// TIA Portal V18 export
// export: Created 2026-06-23T03:11:38.3968089Z, ExportSetting WithDefaults, DisplayName Totally Integrated Automation Portal, DisplayVersion V18, DisplayName TIA Portal Openness, DisplayVersion V18, DisplayName TIA Portal Version Control Interface, DisplayVersion V18, DisplayName STEP 7 Professional, DisplayVersion V18, DisplayName STEP 7 Safety, DisplayVersion V18, DisplayName WinCC Professional, DisplayVersion V18
Screen "Screen_1"  1440x900, Number=2
  ScreenLayer 
    GraphicView "Graphic view_1" at 0,0 size 1440x900  Picture=Thiết kế chưa có tên (2)_1
    GraphicIOField "Graphic I/O field_9" at 430,521 size 275x288  Mode=Output, OnValue=1, PictureList=GL_BonChua_MucDich
      ProcessValue := HMI_Anim_BonChua1_MucDich
    GraphicIOField "Graphic I/O field_10" at 154,90 size 233x295  Mode=Output, OnValue=1, PictureList=GL_BonTron_MucDich
      ProcessValue := HMI_Anim_Bon1_MucDich
    GraphicIOField "Graphic I/O field_2" at 904,517 size 275x288  Mode=Output, OnValue=1, PictureList=GL_BonChua_MucDich
      ProcessValue := HMI_Anim_BonChua2_MucDich
    GraphicIOField "Graphic I/O field_3" at 486,90 size 233x295  Mode=Output, OnValue=1, PictureList=GL_BonTron_MucDich
      ProcessValue := HMI_Anim_Bon2_MucDich
    GraphicIOField "Graphic I/O field_4" at 811,89 size 233x295  Mode=Output, OnValue=1, PictureList=GL_BonTron_MucDich
      ProcessValue := HMI_Anim_Bon4_MucDich
    GraphicIOField "Graphic I/O field_6" at 1160,89 size 233x295  Mode=Output, OnValue=1, PictureList=GL_BonTron_MucDich
      ProcessValue := HMI_Anim_Bon3_MucDich
    GraphicView "Graphic view_3" at 201,61 size 11x113  Picture=Graphic_24
    GraphicIOField "Graphic I/O field_5" at 189,70 size 51x78  Mode=Output, OnValue=1, PictureList=GL_Van_NamDoc
      ProcessValue := V3230_Nuoc_Bon1
    GraphicView "Graphic view_2" at 544,60 size 11x113  Picture=Graphic_24
    GraphicIOField "Graphic I/O field_12" at 533,70 size 51x78  Mode=Output, OnValue=1, PictureList=GL_Van_NamDoc
      ProcessValue := V3235_Nuoc_Bon2
    GraphicView "Graphic view_4" at 869,59 size 11x113  Picture=Graphic_24
    GraphicIOField "Graphic I/O field_13" at 860,69 size 51x78  Mode=Output, OnValue=1, PictureList=GL_Van_NamDoc
      ProcessValue := V3245_Nuoc_Bon4
    GraphicView "Graphic view_5" at 1204,58 size 11x117  Picture=Graphic_24
    GraphicIOField "Graphic I/O field_14" at 1193,67 size 51x78  Mode=Output, OnValue=1, PictureList=GL_Van_NamDoc
      ProcessValue := V3240_Nuoc_Bon3
    GraphicView "Graphic view_6" at 229,330 size 11x172  Picture=Graphic_24
    GraphicIOField "Graphic I/O field_11" at 220,429 size 51x78  Mode=Output, OnValue=1, PictureList=GL_Van_NamDoc
      ProcessValue := V3234_Xa_Bon1
    GraphicIOField "Graphic I/O field_8" at 220,339 size 51x78  Mode=Output, OnValue=1, PictureList=GL_Van_NamDoc
      ProcessValue := V3232_Xa_Bon1
    GraphicView "Graphic view_7" at 568,331 size 11x211  Picture=Graphic_24
    GraphicView "Graphic view_8" at 869,328 size 11x164  Picture=Graphic_24
    GraphicView "Graphic view_9" at 1224,328 size 11x164  Picture=Graphic_24
    GraphicIOField "Graphic I/O field_15" at 556,341 size 51x78  Mode=Output, OnValue=1, PictureList=GL_Van_NamDoc
      ProcessValue := V3237_Xa_Bon2
    GraphicIOField "Graphic I/O field_16" at 558,417 size 51x78  Mode=Output, OnValue=1, PictureList=GL_Van_NamDoc
      ProcessValue := V3239_Xa_Bon2
    GraphicIOField "Graphic I/O field_18" at 857,346 size 51x78  Mode=Output, OnValue=1, PictureList=GL_Van_NamDoc
      ProcessValue := V3247_Xa_Bon4
    GraphicIOField "Graphic I/O field_20" at 857,412 size 51x78  Mode=Output, OnValue=1, PictureList=GL_Van_NamDoc
      ProcessValue := V3249_Xa_Bon4
    GraphicIOField "Graphic I/O field_19" at 1214,347 size 51x78  Mode=Output, OnValue=1, PictureList=GL_Van_NamDoc
      ProcessValue := V3242_Xa_Bon3
    GraphicIOField "Graphic I/O field_21" at 1213,419 size 51x78  Mode=Output, OnValue=1, PictureList=GL_Van_NamDoc
      ProcessValue := V3244_Xa_Bon3
    GraphicView "Graphic view_10" at 223,500 size 25x5  Picture=Graphic_25
    GraphicView "Graphic view_11" at 1216,490 size 25x5  Picture=Graphic_25
    GraphicView "Graphic view_12" at 223,523 size 25x5  Picture=Graphic_25
    GraphicView "Graphic view_13" at 1216,515 size 25x5  Picture=Graphic_25
    GraphicView "Graphic view_14" at 252,501 size 5x26  Picture=Graphic_24
    GraphicView "Graphic view_15" at 1206,492 size 5x26  Picture=Graphic_24
    GraphicView "Graphic view_16" at 254,510 size 242x11  Picture=Graphic_25
    GraphicView "Graphic view_17" at 487,513 size 11x57  Picture=Graphic_24
    GraphicView "Graphic view_18" at 521,159 size 11x19  Picture=Graphic_24
    GraphicView "Graphic view_19" at 440,157 size 90x11  Picture=Graphic_25
    GraphicView "Graphic view_20" at 437,160 size 11x408  Picture=Graphic_24
    GraphicView "Graphic view_21" at 231,560 size 213x11  Picture=Graphic_25
    GraphicView "Graphic view_22" at 228,525 size 11x44  Picture=Graphic_24
    GraphicView "Graphic view_23" at 630,485 size 248x11  Picture=Graphic_25
    GraphicView "Graphic view_24" at 626,488 size 11x75  Picture=Graphic_24
    GraphicView "Graphic view_25" at 640,503 size 11x68  Picture=Graphic_24
    GraphicView "Graphic view_26" at 644,501 size 566x11  Picture=Graphic_25
    GraphicView "Graphic view_27" at 1224,517 size 11x51  Picture=Graphic_24
    GraphicView "Graphic view_28" at 1142,560 size 90x11  Picture=Graphic_25
    GraphicView "Graphic view_29" at 1139,99 size 11x469  Picture=Graphic_24
    GraphicView "Graphic view_30" at 1005,93 size 143x11  Picture=Graphic_25
    GraphicView "Graphic view_31" at 1000,95 size 11x86  Picture=Graphic_24
    GraphicView "Graphic view_32" at 564,755 size 11x103  Picture=Graphic_24
    GraphicIOField "Graphic I/O field_24" at 554,759 size 51x78  Mode=Output, OnValue=1, PictureList=GL_Van_NamDoc
      ProcessValue := V3331_Xa_BonChua1
    GraphicView "Graphic view_33" at 567,849 size 22x11  Picture=Graphic_25
    GraphicView "Graphic view_34" at 581,833 size 11x40  Picture=Graphic_24
    GraphicView "Graphic view_36" at 132,426 size 8x44  Picture=Graphic_28
    GraphicView "Graphic view_35" at 133,425 size 103x6  Picture=Graphic_29
    GraphicIOField "Graphic I/O field_7" at 133,396 size 83x47  Mode=Output, OnValue=1, PictureList=GL_Van_NamNgang
      ProcessValue := V3233_Xa_Bon1
    GraphicIOField "Graphic I/O field_33" at 282,542 size 60x42  Mode=Output, OnValue=1, PictureList=GL_Pump_ChuyenDich
      ProcessValue := Pump3264_Chuyen_Nhanh1
    GraphicView "Graphic view_38" at 371,61 size 2x119  Picture=Graphic_24
    GraphicView "Graphic view_40" at 352,178 size 22x2  Picture=Graphic_25
    GraphicView "Graphic view_39" at 361,99 size 21x47  Picture=Graphic_32
    GraphicView "Graphic view_41" at 125,453 size 21x47  Picture=Graphic_32
    GraphicView "Graphic view_37" at 341,167 size 28x25  Picture=Graphic_34
    GraphicView "Graphic view_42" at 473,422 size 103x6  Picture=Graphic_29
    GraphicIOField "Graphic I/O field_17" at 471,394 size 83x47  Mode=Output, OnValue=1, PictureList=GL_Van_NamNgang
      ProcessValue := V3238_Xa_Bon2
    GraphicView "Graphic view_43" at 472,423 size 8x44  Picture=Graphic_28
    GraphicView "Graphic view_44" at 466,451 size 21x47  Picture=Graphic_32
    GraphicView "Graphic view_45" at 872,415 size 108x6  Picture=Graphic_29
    GraphicIOField "Graphic I/O field_22" at 903,387 size 83x47  Mode=Output, OnValue=1, PictureList=GL_Van_NamNgang
      ProcessValue := V3248_Xa_Bon4
    GraphicView "Graphic view_46" at 976,415 size 8x35  Picture=Graphic_28
    GraphicView "Graphic view_47" at 970,434 size 21x47  Picture=Graphic_32
    GraphicView "Graphic view_48" at 1226,422 size 118x6  Picture=Graphic_29
    GraphicIOField "Graphic I/O field_23" at 1257,394 size 83x47  Mode=Output, OnValue=1, PictureList=GL_Van_NamNgang
      ProcessValue := V3243_Xa_Bon3
    GraphicView "Graphic view_49" at 1336,422 size 8x35  Picture=Graphic_28
    GraphicView "Graphic view_50" at 1331,441 size 21x47  Picture=Graphic_32
    GraphicView "Graphic view_51" at 709,59 size 2x119  Picture=Graphic_24
    GraphicView "Graphic view_52" at 1047,60 size 2x116  Picture=Graphic_24
    GraphicView "Graphic view_53" at 1387,60 size 2x114  Picture=Graphic_24
    GraphicView "Graphic view_54" at 700,102 size 21x47  Picture=Graphic_32
    GraphicView "Graphic view_55" at 1038,104 size 21x47  Picture=Graphic_32
    GraphicView "Graphic view_56" at 1378,106 size 21x47  Picture=Graphic_32
    GraphicView "Graphic view_57" at 689,177 size 22x2  Picture=Graphic_25
    GraphicView "Graphic view_58" at 1016,175 size 33x2  Picture=Graphic_25
    GraphicView "Graphic view_59" at 1366,173 size 22x2  Picture=Graphic_25
    GraphicView "Graphic view_60" at 672,166 size 28x25  Picture=Graphic_34
    GraphicView "Graphic view_61" at 1000,165 size 28x25  Picture=Graphic_34
    GraphicView "Graphic view_62" at 1347,162 size 28x25  Picture=Graphic_34
    GraphicView "Graphic view_63" at 584,865 size 16x11  Picture=Graphic_25
    GraphicView "Graphic view_64" at 584,830 size 159x11  Picture=Graphic_25
    GraphicView "Graphic view_65" at 598,858 size 5x26  Picture=Graphic_24
    GraphicView "Graphic view_66" at 603,858 size 5x26  Picture=Graphic_24
    GraphicView "Graphic view_67" at 605,866 size 68x11  Picture=Graphic_25
    GraphicIOField "Graphic I/O field_1" at 608,851 size 60x42  Mode=Output, OnValue=1, PictureList=GL_Pump_ChuyenDich
      ProcessValue := Pump3362_Xa_BonChua1
    GraphicView "Graphic view_68" at 668,858 size 5x26  Picture=Graphic_24
    GraphicView "Graphic view_69" at 674,858 size 5x26  Picture=Graphic_24
    GraphicView "Graphic view_70" at 675,866 size 13x11  Picture=Graphic_25
    GraphicView "Graphic view_71" at 682,513 size 11x361  Picture=Graphic_24
    GraphicIOField "Graphic I/O field_25" at 672,597 size 51x78  Mode=Output, OnValue=1, PictureList=GL_Van_NamDoc
      ProcessValue := V3334_DieuHuong_BonChua1
    GraphicView "Graphic view_72" at 684,510 size 376x11  Picture=Graphic_25
    GraphicView "Graphic view_73" at 1053,512 size 11x26  Picture=Graphic_24
    GraphicIOField "Graphic I/O field_34" at 587,792 size 90x71  Mode=Output, OnValue=1, PictureList=GL_Pump_TuanHoanLoc
      ProcessValue := Pump3361_LuanChuyen_BonChua1
    GraphicView "Graphic view_74" at 735,752 size 11x144  Picture=Graphic_24
    GraphicIOField "Graphic I/O field_27" at 725,822 size 51x78  Mode=Output, OnValue=1, PictureList=GL_Van_NamDoc
      ProcessValue := V3333_DieuHuong_BonChua1
    GraphicIOField "Graphic I/O field_26" at 725,757 size 51x78  Mode=Output, OnValue=1, PictureList=GL_Van_NamDoc
      ProcessValue := V3335_DieuHuong_BonChua1
    GraphicView "Graphic view_75" at 739,889 size 528x11  Picture=Graphic_25
    GraphicView "Graphic view_76" at 738,748 size 65x11  Picture=Graphic_25
    GraphicView "Graphic view_77" at 799,521 size 11x236  Picture=Graphic_24
    GraphicView "Graphic view_78" at 801,518 size 211x11  Picture=Graphic_25
    GraphicView "Graphic view_79" at 1005,520 size 11x38  Picture=Graphic_24
    GraphicView "Graphic view_80" at 469,833 size 103x6  Picture=Graphic_29
    GraphicView "Graphic view_81" at 467,834 size 8x44  Picture=Graphic_28
    GraphicView "Graphic view_82" at 461,853 size 21x47  Picture=Graphic_32
    GraphicIOField "Graphic I/O field_30" at 467,804 size 83x47  Mode=Output, OnValue=1, PictureList=GL_Van_NamNgang
      ProcessValue := V3332_Xa_BonChua1
    GraphicView "Graphic view_83" at 1040,751 size 11x75  Picture=Graphic_24
    GraphicIOField "Graphic I/O field_28" at 1030,754 size 51x78  Mode=Output, OnValue=1, PictureList=GL_Van_NamDoc
      ProcessValue := V3338_Xa_BonChua2
    GraphicView "Graphic view_84" at 1042,818 size 62x11  Picture=Graphic_25
    GraphicView "Graphic view_85" at 1100,802 size 11x40  Picture=Graphic_24
    GraphicView "Graphic view_86" at 1104,800 size 103x11  Picture=Graphic_25
    GraphicIOField "Graphic I/O field_35" at 1108,764 size 90x71  Mode=Output, OnValue=1, PictureList=GL_Pump_TuanHoanLoc
      ProcessValue := Pump3364_Filter
    GraphicView "Graphic view_87" at 1103,833 size 12x11  Picture=Graphic_25
    GraphicView "Graphic view_88" at 1112,825 size 5x26  Picture=Graphic_24
    GraphicView "Graphic view_89" at 1117,825 size 5x26  Picture=Graphic_24
    GraphicView "Graphic view_90" at 1118,833 size 72x11  Picture=Graphic_25
    GraphicIOField "Graphic I/O field_36" at 1123,820 size 60x42  Mode=Output, OnValue=1, PictureList=GL_Pump_ChuyenDich
      ProcessValue := Pump3365_Filter
    GraphicView "Graphic view_91" at 1186,825 size 5x26  Picture=Graphic_24
    GraphicView "Graphic view_92" at 1192,825 size 5x26  Picture=Graphic_24
    GraphicView "Graphic view_93" at 1195,833 size 13x11  Picture=Graphic_25
    GraphicView "Graphic view_94" at 1201,589 size 11x252  Picture=Graphic_24
    GraphicIOField "Graphic I/O field_29" at 1191,655 size 51x78  Mode=Output, OnValue=1, PictureList=GL_Van_NamDoc
      ProcessValue := V3341_Duong_Filter
    GraphicIOField "Graphic I/O field_37" at 1156,541 size 60x42  Mode=Output, OnValue=1, PictureList=GL_Pump_ChuyenDich
      ProcessValue := Pump3265_Chuyen_Nhanh2
    GraphicView "Graphic view_95" at 1204,587 size 150x11  Picture=Graphic_25
    GraphicView "Graphic view_96" at 1257,590 size 11x307  Picture=Graphic_24
    GraphicView "Graphic view_97" at 1345,589 size 11x192  Picture=Graphic_24
    GraphicView "Graphic view_98" at 1352,589 size 75x6  Picture=Graphic_29
    GraphicIOField "Graphic I/O field_32" at 1346,558 size 83x47  Mode=Output, OnValue=1, PictureList=GL_Van_NamNgang
      ProcessValue := V3340_Duong_Filter
    GraphicView "Graphic view_99" at 1420,591 size 8x35  Picture=Graphic_28
    GraphicView "Graphic view_100" at 1414,607 size 21x47  Picture=Graphic_32
    GraphicView "Graphic view_102" at 1368,50 size 41x72  Picture=Graphic_37
    GraphicView "Graphic view_103" at 1365,159 size 28x31  Picture=Graphic_38
    GraphicView "Graphic view_104" at 1027,50 size 41x72  Picture=Graphic_37
    GraphicView "Graphic view_105" at 690,50 size 41x72  Picture=Graphic_37
    GraphicView "Graphic view_106" at 352,50 size 41x72  Picture=Graphic_37
    GraphicView "Graphic view_107" at 352,121 size 41x74  Picture=Graphic_39
    GraphicView "Graphic view_108" at 691,121 size 41x74  Picture=Graphic_39
    GraphicView "Graphic view_109" at 1028,121 size 41x74  Picture=Graphic_39
    GraphicView "Graphic view_110" at 1368,119 size 41x74  Picture=Graphic_39
    GraphicView "Graphic view_101" at 1012,165 size 45x26  Picture=Graphic_40
    GraphicView "Graphic view_111" at 676,167 size 45x26  Picture=Graphic_40
    GraphicView "Graphic view_112" at 341,167 size 38x26  Picture=Graphic_40
    GraphicIOField "Graphic I/O field_38" at 123,84 size 292x298  Mode=Output, OnValue=1, PictureList=GL_Khuay_8Frame
      ProcessValue := HMI_Anim_Bon1_Frame
    GraphicIOField "Graphic I/O field_39" at 459,83 size 292x298  Mode=Output, OnValue=1, PictureList=GL_Khuay_8Frame
      ProcessValue := HMI_Anim_Bon2_Frame
    GraphicIOField "Graphic I/O field_40" at 782,86 size 292x298  Mode=Output, OnValue=1, PictureList=GL_Khuay_8Frame
      ProcessValue := HMI_Anim_Bon4_Frame
    GraphicIOField "Graphic I/O field_41" at 1130,90 size 292x298  Mode=Output, OnValue=1, PictureList=GL_Khuay_8Frame
      ProcessValue := HMI_Anim_Bon3_Frame
    GraphicView "Graphic view_113" at 1280,567 size 56x45  Picture=Graphic_44
    GraphicView "Graphic view_115" at 1338,606 size 28x43  Picture=Graphic_46
    GraphicView "Graphic view_114" at 1246,722 size 28x43  Picture=Graphic_46
    GraphicView "Graphic view_116" at 1340,714 size 33x47  Picture=Graphic_47
    GraphicView "Graphic view_117" at 1327,779 size 50x52  Picture=Graphic_48
    GraphicView "Graphic view_118" at 1341,815 size 21x47  Picture=Graphic_32
    GraphicView "Graphic view_119" at 1337,843 size 29x56  Picture=Graphic_49
    GraphicView "Graphic view_120" at 939,821 size 108x6  Picture=Graphic_29
    GraphicIOField "Graphic I/O field_31" at 930,792 size 83x47  Mode=Output, OnValue=1, PictureList=GL_Van_NamNgang
      ProcessValue := V3339_Xa_BonChua2
    GraphicView "Graphic view_121" at 934,821 size 8x44  Picture=Graphic_28
    GraphicView "Graphic view_122" at 929,842 size 21x47  Picture=Graphic_32
    IOField "I/O field_1" at 133,61 size 47x32  DataFormat=Decimal, FormatPattern=999.9, Mode=InOutput
      ProcessValue := FQ3200_Bon1_Eff
    GraphicView "Graphic view_123" at 775,636 size 55x48  Picture=Graphic_50
    IOField "I/O field_2" at 300,127 size 43x28  DataFormat=Decimal, FormatPattern=999.9, Mode=InOutput
      ProcessValue := LT3203_Bon1_Eff
    GraphicView "Graphic view_124" at 814,628 size 69x36  Picture=Graphic_51
    GraphicView "Graphic view_125" at 858,575 size 22x78  Picture=Graphic_39
    GraphicView "Graphic view_126" at 858,516 size 22x85  Picture=Graphic_39
    GraphicView "Graphic view_127" at 815,661 size 69x36  Picture=Graphic_51
    GraphicView "Graphic view_128" at 858,671 size 22x85  Picture=Graphic_39
    IOField "I/O field_3" at 832,741 size 51x28  DataFormat=Decimal, FormatPattern=999.9, Mode=InOutput
      ProcessValue := CV3304_Nuoc_Lam_Mat_M
    IOField "I/O field_4" at 791,589 size 44x28  DataFormat=Decimal, FormatPattern=99.9, Mode=InOutput
      ProcessValue := TT3303_TraoDoiNhiet_Eff
    IOField "I/O field_5" at 353,195 size 43x28  DataFormat=Decimal, FormatPattern=99.9, Mode=InOutput
      ProcessValue := TT3204_Bon1_Eff
    IOField "I/O field_6" at 354,296 size 43x28  DataFormat=Decimal, FormatPattern=999.9, Mode=InOutput
      ProcessValue := CV3201_Nuoc_Bon1_M
    IOField "I/O field_7" at 486,65 size 43x28  DataFormat=Decimal, FormatPattern=999.9, Mode=InOutput
      ProcessValue := FQ3205_Bon2_Eff
    IOField "I/O field_8" at 636,129 size 43x28  DataFormat=Decimal, FormatPattern=999.9, Mode=InOutput
      ProcessValue := LT3209_Bon2_Eff
    IOField "I/O field_9" at 689,192 size 43x28  DataFormat=Decimal, FormatPattern=99.9, Mode=InOutput
      ProcessValue := TT3208_Bon2_Eff
    IOField "I/O field_10" at 688,294 size 43x28  DataFormat=Decimal, FormatPattern=999.9, Mode=InOutput
      ProcessValue := CV3206_Hoi_Bon2_M
    IOField "I/O field_11" at 804,61 size 43x28  DataFormat=Decimal, FormatPattern=999.9, Mode=InOutput
      ProcessValue := FQ3215_Bon4_Eff
    IOField "I/O field_12" at 965,127 size 43x28  DataFormat=Decimal, FormatPattern=999.9, Mode=InOutput
      ProcessValue := LT3218_Bon4_Eff
    IOField "I/O field_13" at 1016,190 size 43x28  DataFormat=Decimal, FormatPattern=99.9, Mode=InOutput
      ProcessValue := TT3219_Bon4_Eff
    IOField "I/O field_14" at 1015,293 size 43x28  DataFormat=Decimal, FormatPattern=999.9, Mode=InOutput
      ProcessValue := CV3216_Hoi_Bon4_M
    IOField "I/O field_15" at 1143,62 size 43x28  DataFormat=Decimal, FormatPattern=999.9, Mode=InOutput
      ProcessValue := FQ3210_Bon3_Eff
    IOField "I/O field_16" at 1318,130 size 43x28  DataFormat=Decimal, FormatPattern=999.9, Mode=InOutput
      ProcessValue := LT3213_Bon3_Eff
    IOField "I/O field_17" at 1365,193 size 43x28  DataFormat=Decimal, FormatPattern=99.9, Mode=InOutput
      ProcessValue := TT3214_Bon3_Eff
    IOField "I/O field_18" at 1367,293 size 43x28  DataFormat=Decimal, FormatPattern=999.9, Mode=InOutput
      ProcessValue := CV3211_Nuoc_Bon3_M
    IOField "I/O field_19" at 412,586 size 43x28  DataFormat=Decimal, FormatPattern=999.9, Mode=InOutput
      ProcessValue := LT3302_BonChua1_Eff
    IOField "I/O field_20" at 417,713 size 43x28  DataFormat=Decimal, FormatPattern=99.9, Mode=InOutput
      ProcessValue := TT3301_BonChua1_Eff
    IOField "I/O field_21" at 1134,711 size 43x28  DataFormat=Decimal, FormatPattern=99.9, Mode=InOutput
      ProcessValue := TT3306_BonChua2_Eff
    IOField "I/O field_22" at 1135,589 size 43x28  DataFormat=Decimal, FormatPattern=999.9, Mode=InOutput
      ProcessValue := LT3307_BonChua2_Eff
    IOField "I/O field_23" at 1280,616 size 43x28  DataFormat=Decimal, FormatPattern=99.9, Mode=InOutput
      ProcessValue := PI3308_Truoc_Filter_Eff
    IOField "I/O field_24" at 1280,670 size 43x28  DataFormat=Decimal, FormatPattern=999.9, Mode=InOutput
      ProcessValue := FT3309_Xa_Thanh_Pham_Eff
    TextField "Text field_1" at 183,66 size 16x24  Text="L"
    TextField "Text field_2" at 344,130 size 25x24  Text="%"
    TextField "Text field_3" at 529,67 size 16x24  Text="L"
    TextField "Text field_4" at 848,64 size 16x24  Text="L"
    TextField "Text field_5" at 1187,64 size 16x24  Text="L"
    TextField "Text field_6" at 680,132 size 25x24  Text="%"
    TextField "Text field_7" at 1009,129 size 25x24  Text="%"
    TextField "Text field_8" at 1361,131 size 25x24  Text="%"
    TextField "Text field_9" at 397,198 size 16x24  Text="L"
    TextField "Text field_10" at 734,196 size 16x24  Text="L"
    TextField "Text field_11" at 1061,194 size 16x24  Text="L"
    TextField "Text field_12" at 1410,195 size 16x24  Text="L"
    TextField "Text field_13" at 400,300 size 25x24  Text="°C"
    TextField "Text field_14" at 735,296 size 25x24  Text="°C"
    TextField "Text field_15" at 1061,297 size 25x24  Text="°C"
    TextField "Text field_16" at 1412,296 size 25x24  Text="°C"
    TextField "Text field_17" at 456,589 size 16x24  Text="L"
    TextField "Text field_18" at 462,715 size 16x24  Text="L"
    TextField "Text field_19" at 836,592 size 25x24  Text="°C"
    TextField "Text field_20" at 884,744 size 25x24  Text="%"
    TextField "Text field_21" at 1179,592 size 16x24  Text="L"
    TextField "Text field_22" at 1178,714 size 16x24  Text="L"
    TextField "Text field_23" at 1325,673 size 16x24  Text="L"
    TextField "Text field_24" at 1324,619 size 16x24  Text="L"
    TextField "Text field_25" at 210,58 size 72x22  Text="FT 32.00"
    TextField "Text field_26" at 294,105 size 74x22  Text="CV 32.01"
    TextField "Text field_27" at 128,124 size 60x22  Text="V32.30"
    TextField "Text field_28" at 354,223 size 72x22  Text="LT 32.03"
    TextField "Text field_29" at 355,271 size 72x22  Text="TT 32.04"
    TextField "Text field_30" at 475,117 size 60x22  Text="V32.35"
    TextField "Text field_31" at 554,67 size 72x22  Text="FT 32.05"
    TextField "Text field_32" at 628,108 size 70x22  Text="CV32.06"
    TextField "Text field_33" at 689,221 size 72x22  Text="LT 32.09"
    TextField "Text field_34" at 689,269 size 72x22  Text="TT 32.08"
    TextField "Text field_35" at 1014,218 size 72x22  Text="LT 32.18"
    TextField "Text field_36" at 1015,270 size 72x22  Text="TT 32.19"
    TextField "Text field_37" at 962,99 size 70x22  Text="CV32.16"
    TextField "Text field_38" at 880,64 size 72x22  Text="FT 32.15"
    TextField "Text field_39" at 801,117 size 60x22  Text="V32.45"
    TextField "Text field_40" at 1215,57 size 72x22  Text="FT 32.10"
    TextField "Text field_41" at 1308,110 size 70x22  Text="CV32.11"
    TextField "Text field_42" at 1362,222 size 72x22  Text="LT 32.13"
    TextField "Text field_43" at 1363,268 size 72x22  Text="TT 32.14"
    TextField "Text field_44" at 265,371 size 60x22  Text="V32.32"
    TextField "Text field_45" at 144,435 size 60x22  Text="V32.33"
    TextField "Text field_46" at 271,457 size 60x22  Text="V32.34"
    TextField "Text field_47" at 489,433 size 60x22  Text="V32.38"
    TextField "Text field_48" at 599,371 size 60x22  Text="V32.37"
    TextField "Text field_49" at 603,441 size 60x22  Text="V32.39"
    TextField "Text field_50" at 800,370 size 60x22  Text="V32.47"
    TextField "Text field_51" at 803,437 size 60x22  Text="V32.49"
    TextField "Text field_52" at 963,389 size 60x22  Text="V32.48"
    TextField "Text field_53" at 1164,370 size 60x22  Text="V32.42"
    TextField "Text field_54" at 1157,443 size 60x22  Text="V32.44"
    TextField "Text field_55" at 1317,389 size 60x22  Text="V32.43"
    TextField "Text field_56" at 1359,537 size 60x22  Text="V33.40"
    TextField "Text field_57" at 1184,653 size 60x22  Text="V33.41"
    TextField "Text field_58" at 977,765 size 60x22  Text="V33.38"
    TextField "Text field_59" at 891,797 size 60x22  Text="V33.39"
    TextField "Text field_60" at 768,861 size 60x22  Text="V33.33"
    TextField "Text field_61" at 768,789 size 60x22  Text="V33.35"
    TextField "Text field_62" at 701,653 size 60x22  Text="V33.34"
    TextField "Text field_63" at 484,848 size 60x22  Text="V33.32"
    TextField "Text field_64" at 504,768 size 60x22  Text="V33.31"
    TextField "Text field_65" at 342,339 size 70x29  Text="BỒN 1"
    TextField "Text field_66" at 669,331 size 70x29  Text="BỒN 2"
    TextField "Text field_67" at 998,324 size 70x29  Text="BỒN 4"
    TextField "Text field_68" at 1344,330 size 70x29  Text="BỒN 3"
    TextField "Text field_69" at 1299,474 size 79x29  Text="FILLER"
    TextField "Text field_70" at 1355,671 size 72x22  Text="FT 33.09"
    TextField "Text field_71" at 399,619 size 72x22  Text="LT 32.02"
    TextField "Text field_72" at 399,684 size 72x22  Text="TT 33.01"
    TextField "Text field_73" at 782,568 size 72x22  Text="TT 33.03"
    TextField "Text field_74" at 830,767 size 74x22  Text="CV 33.04"
    TextField "Text field_75" at 1135,614 size 72x22  Text="LT 33.07"
    TextField "Text field_76" at 1129,689 size 68x22  Text="TT33.06"
    TextField "Text field_77" at 1275,643 size 71x22  Text="PI 33.08"
    TextField "Text field_78" at 1275,765 size 59x15  Text="LSH 33.10"
    TextField "Text field_79" at 1277,823 size 59x15  Text="LSH 33.11"
    TextField "Text field_80" at 1357,756 size 83x22  Text="CV FILLER"
    TextField "Text field_81" at 283,582 size 71x17  Text="PUMP 32.64"
    TextField "Text field_82" at 601,794 size 71x17  Text="PUMP 33.61"
    TextField "Text field_83" at 608,843 size 71x17  Text="PUMP 33.62"
    TextField "Text field_84" at 1110,765 size 71x17  Text="PUMP 33.64"
    TextField "Text field_85" at 1139,859 size 71x17  Text="PUMP 33.65"
    TextField "Text field_86" at 1149,531 size 71x17  Text="PUMP 32.65"
    TextField "Text field_87" at 1260,546 size 102x22  Text="CPP FILLTER"
